FUNCTION_BLOCK FB_ErrorBuffer
VAR
	fbMemRingBuffer : FB_MemRingBuffer;
	BufferArray  : ARRAY [0..100] OF BYTE;
END_VAR

METHOD PUBLIC AddErrorMessage
VAR_INPUT
	eErrorMessage : REFERENCE TO eErrorList;
END_VAR
fbMemRingBuffer.A_AddTail(	pWrite := ADR(eErrorMessage),
							cbWrite := SIZEOF(eErrorMessage),
							pBuffer := ADR(BufferArray),
							cbBuffer := SIZEOF(BufferArray));
END_METHOD

METHOD PUBLIC GetAndRemoveErrorMessage
VAR_OUTPUT
	eErrorMessage : eErrorList;
END_VAR
fbMemRingBuffer.A_RemoveHead(	pRead := ADR(eErrorMessage),
								cbRead := SIZEOF(eErrorMessage),
								pBuffer := ADR(BufferArray),
								cbBuffer := SIZEOF(BufferArray));
END_METHOD

PROPERTY getNumberOfMessages : UDINT
GET
getNumberOfMessages := fbMemRingBuffer.nCount;
END_GET
END_PROPERTY

END_FUNCTION_BLOCK

(* stored: Version 1.1.0.1, ProductVersion 3.1.4024.12
   POU FB_ErrorBuffer: Id {0eb830b0-ad0d-4933-8fc2-da6936ba2c06}, SpecialFunc None
   Method AddErrorMessage: Id {e698bc52-df31-43c0-876d-940714f97c03}
   Method GetAndRemoveErrorMessage: Id {b7bcbfb8-e01e-45ce-88b4-f3b1aa515d62}
   Property getNumberOfMessages: Id {e53906eb-2cc9-4439-ab52-c8aed52e6ca2}
   Get Get: Id {5efdc35b-72aa-4285-995a-6f82112207ac} *)
